{attribute addProperty BoxType "EPP1816-3008-0016"}
{attribute addProperty Id "DIG_Inputs_ChannelAT %I*ARRAY[0..1] OF DIG_Inputs_Channel_628B507D128160AI_Inputs_ChannelAT %I*ARRAY[0..5] OF AI_Inputs_Channel_36527000192240DIG_Inputs_DeviceAT %I*DIG_Inputs_Device_5061D9393240WcStateAT %I*WcState_F855686C1620InfoDataAT %I*InfoData_BC63D37F80100"}
{attribute addProperty CRC "3082739873"}
{attribute addProperty SizeInBites "448"}
{attribute addProperty SizeInBytes "56"}
TYPE EPP1816_5F09590E :
STRUCT
	{attribute addProperty Name "DIG_Inputs_Channel"}
	DIG_Inputs_Channel : ARRAY[0..1] OF DIG_Inputs_Channel_628B507D;
	{attribute addProperty Name "AI_Inputs_Channel"}
	AI_Inputs_Channel : ARRAY[0..5] OF AI_Inputs_Channel_36527000;
	{attribute addProperty Name "DIG_Inputs_Device"}
	DIG_Inputs_Device : DIG_Inputs_Device_5061D939;
	{attribute addProperty Name "WcState"}
	WcState : WcState_F855686C;
	{attribute addProperty Name "InfoData"}
	InfoData : InfoData_BC63D37F;
END_STRUCT
END_TYPE

(* stored: Version 1.2.0.0, ProductVersion 3.1.4024.9
   DUT EPP1816_5F09590E: Id {f3c046d8-2c39-4871-944f-c2bf722c5841} *)
